// TIA Portal V18 export
FUNCTION "FC_AnalogInCoverter" : Void   // FC7, STL
{ S7_Optimized_Access := 'TRUE' }
VERSION : 0.1
// stored: AutoNumber true, UDAEnableTagReadback false
   VAR_INPUT
      in_AnalogData : Int;
      in_ScaleMax : Real;
      in_SacaleMin : Real;
   END_VAR
   VAR_OUTPUT
      out_AnalogData : Real;
   END_VAR
   VAR_TEMP
      normData : Real;
   END_VAR
BEGIN

NETWORK
TITLE = 
//Conversor de entradas analogicas
      CALL  NORM_X
      ( MIN     := 0,
        VALUE   := #in_AnalogData,
        MAX     := 27468,
        Ret_Val := #normData
      );

      CALL  SCALE_X
      ( MIN     := #in_SacaleMin,
        VALUE   := #normData,
        MAX     := #in_ScaleMax,
        Ret_Val := #out_AnalogData
      );


END_FUNCTION
